Universal Robots PolyScope program: roller scanner.urp

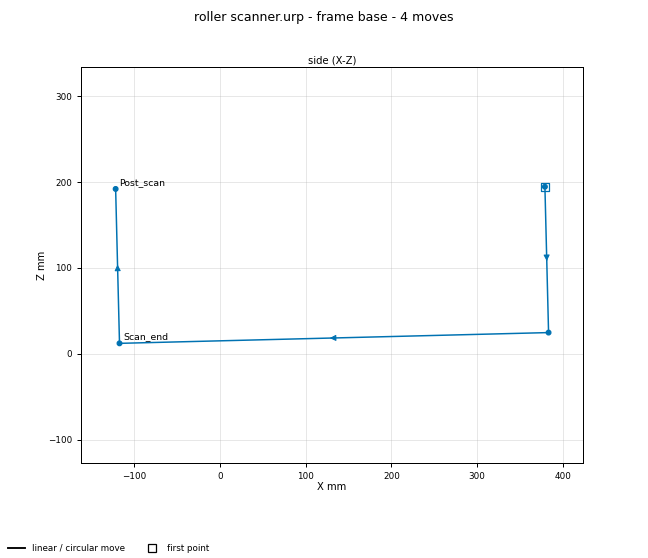
[picture p0: tool path of roller scanner.urp in frame base, 4 of 4 moves have a stored position in this frame; points joined in program order, loops and branches not executed]
Program roller scanner (createdIn=3.2.18654 lastSavedIn=3.2.18654 directory=/home/ur/ursim-3.2/programs installation=default robotSerialNumber=2014359999)
Calibrated DH parameters: a=[0, -0.425, -0.39225, 0, 0, 0]; d=[0.089159, 0, 0, 0.10915, 0.09465, 0.0823]; alpha=[1.570796, 0, 0, 1.570796, -1.570796, 0]; deltaTheta=[0, 0, 0, 0, 0, 0]
Robot Program (runOnlyOnce=false motionType=MoveJ speed=1.047198 acceleration=1.396263 recalculateMotions=false)
  MoveJ speed 60 deg/s, acceleration 80 deg/s^2 (recalculateMotions=false)
    Waypoint Pre_scan: TCP in base x=378.827 y=-432.427 z=194.607 mm, rx=-0.0012 ry=3.1163 rz=0.0389 rad; joints [-38.129, -109.378, -103.622, -56.754, 92.012, 51.831] deg
  MoveL speed 250 mm/s, acceleration 1200 mm/s^2 (recalculateMotions=false) feature=Base
    Waypoint Scan_start: TCP in base x=383.087 y=-428.183 z=24.714 mm, rx=-0.0012 ry=3.1163 rz=0.0389 rad; joints [-37.523, -126.188, -109.933, -33.612, 92.009, 52.437] deg
  MoveL speed 250 mm/s, acceleration 1200 mm/s^2 (recalculateMotions=false) feature=Base
    Waypoint Scan_end: TCP in base x=-116.756 y=-428.418 z=12.175 mm, rx=-0.0012 ry=3.1163 rz=0.0389 rad; joints [-91.283, -118.123, -131.267, -22.073, 91.403, -1.346] deg
  MoveL speed 250 mm/s, acceleration 1200 mm/s^2 (recalculateMotions=false) feature=Base
    Waypoint Post_scan: TCP in base x=-121.266 y=-432.912 z=192.062 mm, rx=-0.0012 ry=3.1163 rz=0.0389 rad; joints [-91.859, -94.185, -122.854, -54.438, 91.389, -1.922] deg
